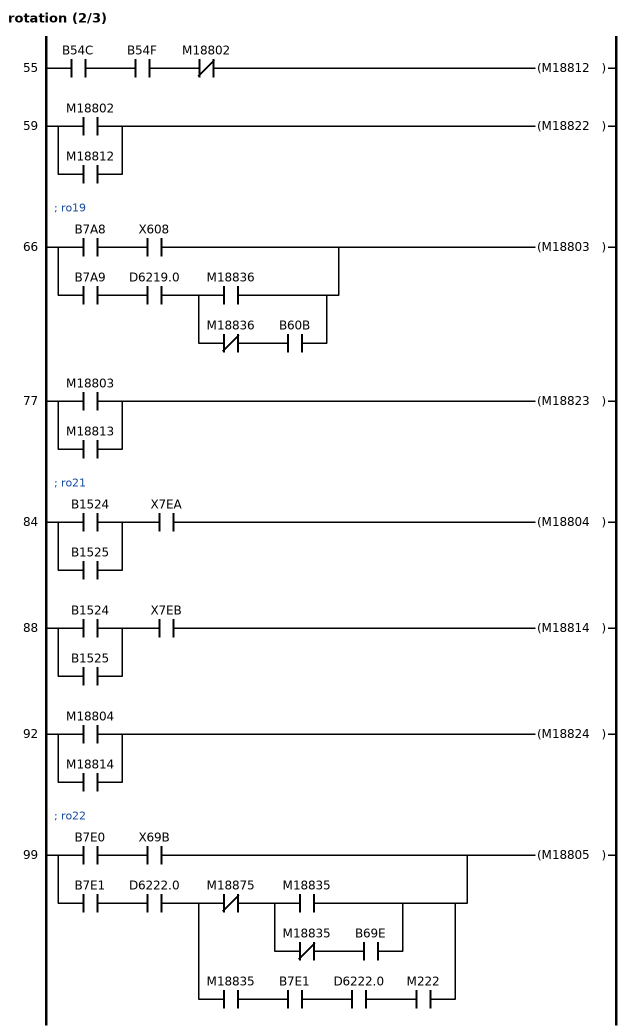
55    LD      B54C
      AND     B54F
      ANI     M18802
      OUT     M18812
59    LD      M18802
      OR      M18812
      OUT     M18822
; ro19
66    LD      B7A8
      AND     X608
      LD      B7A9
      AND     D6219.0
      LD      M18836
      LDI     M18836
      AND     B60B
      ORB
      ANB
      ORB
      OUT     M18803
77    LD      M18803
      OR      M18813
      OUT     M18823
; ro21
84    LD      B1524
      OR      B1525
      AND     X7EA
      OUT     M18804
88    LD      B1524
      OR      B1525
      AND     X7EB
      OUT     M18814
92    LD      M18804
      OR      M18814
      OUT     M18824
; ro22
99    LD      B7E0
      AND     X69B
      LD      B7E1
      AND     D6222.0
      LDI     M18875
      LD      M18835
      LDI     M18835
      AND     B69E
      ORB
      ANB
      LD      M18835
      AND     B7E1
      AND     D6222.0
      AND     M222
      ORB
      ANB
      ORB
      OUT     M18805
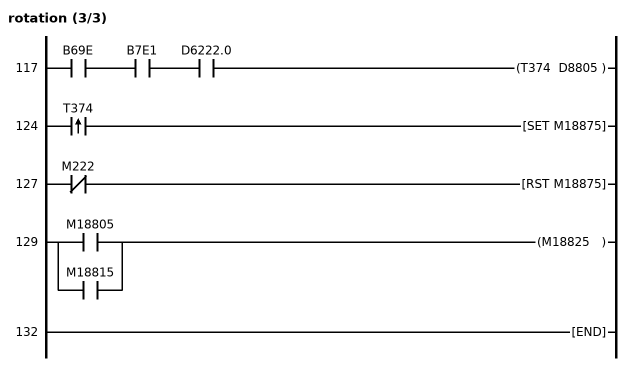
117   LD      B69E
      AND     B7E1
      AND     D6222.0
      OUT     T374 D8805
124   LDP     T374
      SET     M18875
127   LDI     M222
      RST     M18875
129   LD      M18805
      OR      M18815
      OUT     M18825
132   END
END_PROGRAM

PROGRAM safty
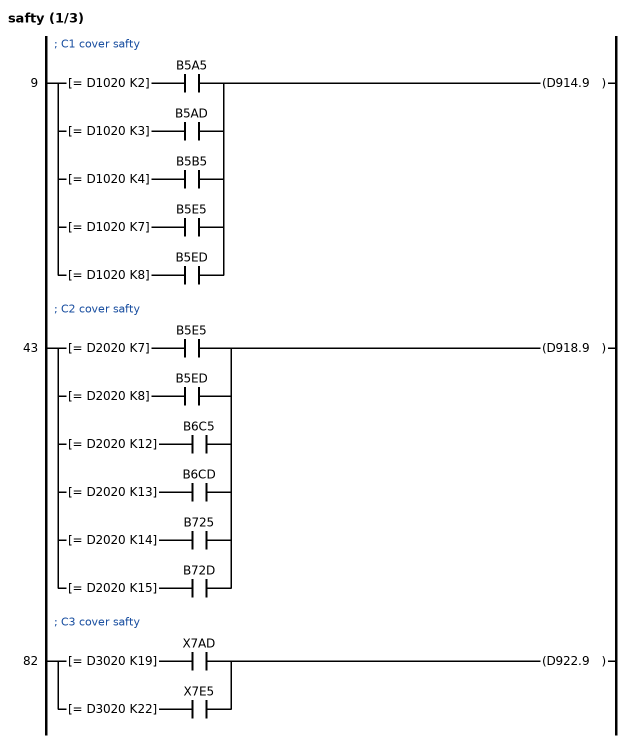
; C1 cover safty
9     LD=     D1020 K2
      AND     B5A5
      LD=     D1020 K3
      AND     B5AD
      ORB
      LD=     D1020 K4
      AND     B5B5
      ORB
      LD=     D1020 K7
      AND     B5E5
      ORB
      LD=     D1020 K8
      AND     B5ED
      ORB
      OUT     D914.9
; C2 cover safty
43    LD=     D2020 K7
      AND     B5E5
      LD=     D2020 K8
      AND     B5ED
      ORB
      LD=     D2020 K12
      AND     B6C5
      ORB
      LD=     D2020 K13
      AND     B6CD
      ORB
      LD=     D2020 K14
      AND     B725
      ORB
      LD=     D2020 K15
      AND     B72D
      ORB
      OUT     D918.9
; C3 cover safty
82    LD=     D3020 K19
      AND     X7AD
      LD=     D3020 K22
      AND     X7E5
      ORB
      OUT     D922.9
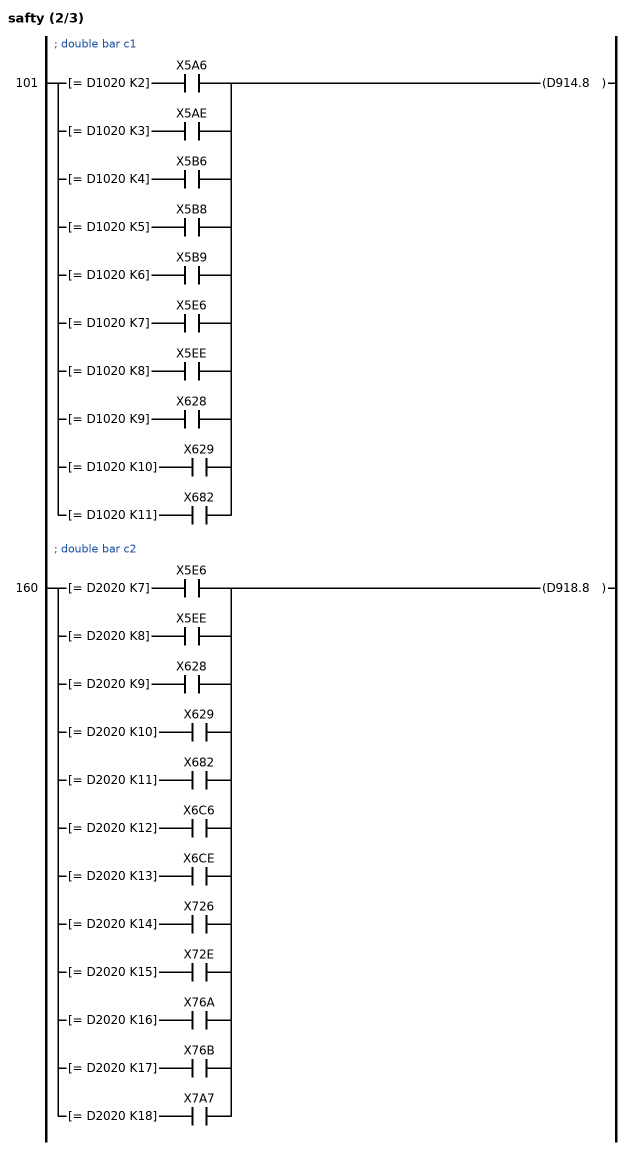
; double bar c1
101   LD=     D1020 K2
      AND     X5A6
      LD=     D1020 K3
      AND     X5AE
      ORB
      LD=     D1020 K4
      AND     X5B6
      ORB
      LD=     D1020 K5
      AND     X5B8
      ORB
      LD=     D1020 K6
      AND     X5B9
      ORB
      LD=     D1020 K7
      AND     X5E6
      ORB
      LD=     D1020 K8
      AND     X5EE
      ORB
      LD=     D1020 K9
      AND     X628
      ORB
      LD=     D1020 K10
      AND     X629
      ORB
      LD=     D1020 K11
      AND     X682
      ORB
      OUT     D914.8
; double bar c2
160   LD=     D2020 K7
      AND     X5E6
      LD=     D2020 K8
      AND     X5EE
      ORB
      LD=     D2020 K9
      AND     X628
      ORB
      LD=     D2020 K10
      AND     X629
      ORB
      LD=     D2020 K11
      AND     X682
      ORB
      LD=     D2020 K12
      AND     X6C6
      ORB
      LD=     D2020 K13
      AND     X6CE
      ORB
      LD=     D2020 K14
      AND     X726
      ORB
      LD=     D2020 K15
      AND     X72E
      ORB
      LD=     D2020 K16
      AND     X76A
      ORB
      LD=     D2020 K17
      AND     X76B
      ORB
      LD=     D2020 K18
      AND     X7A7
      ORB
      OUT     D918.8
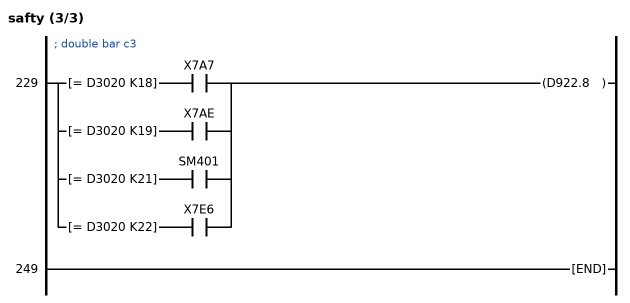
; double bar c3
229   LD=     D3020 K18
      AND     X7A7
      LD=     D3020 K19
      AND     X7AE
      ORB
      LD=     D3020 K21
      AND     SM401
      ORB
      LD=     D3020 K22
      AND     X7E6
      ORB
      OUT     D922.8
249   END
END_PROGRAM

PROGRAM Scrubber
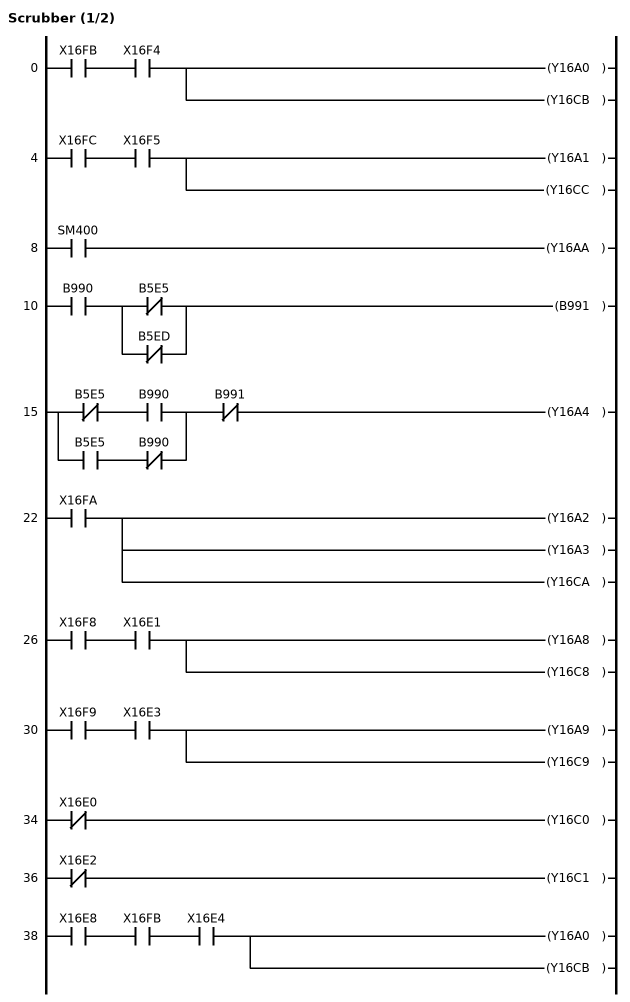
0     LD      X16FB
      AND     X16F4
      OUT     Y16A0
      OUT     Y16CB
4     LD      X16FC
      AND     X16F5
      OUT     Y16A1
      OUT     Y16CC
8     LD      SM400
      OUT     Y16AA
10    LD      B990
      LDI     B5E5
      ORI     B5ED
      ANB
      OUT     B991
15    LDI     B5E5
      AND     B990
      LD      B5E5
      ANI     B990
      ORB
      ANI     B991
      OUT     Y16A4
22    LD      X16FA
      OUT     Y16A2
      OUT     Y16A3
      OUT     Y16CA
26    LD      X16F8
      AND     X16E1
      OUT     Y16A8
      OUT     Y16C8
30    LD      X16F9
      AND     X16E3
      OUT     Y16A9
      OUT     Y16C9
34    LDI     X16E0
      OUT     Y16C0
36    LDI     X16E2
      OUT     Y16C1
38    LD      X16E8
      AND     X16FB
      AND     X16E4
      OUT     Y16A0
      OUT     Y16CB
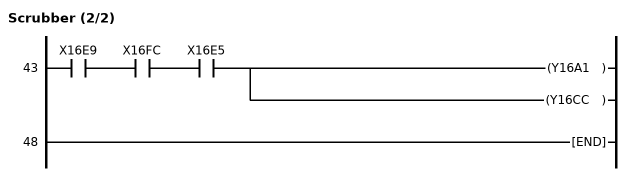
43    LD      X16E9
      AND     X16FC
      AND     X16E5
      OUT     Y16A1
      OUT     Y16CC
48    END
END_PROGRAM

PROGRAM send_to_c
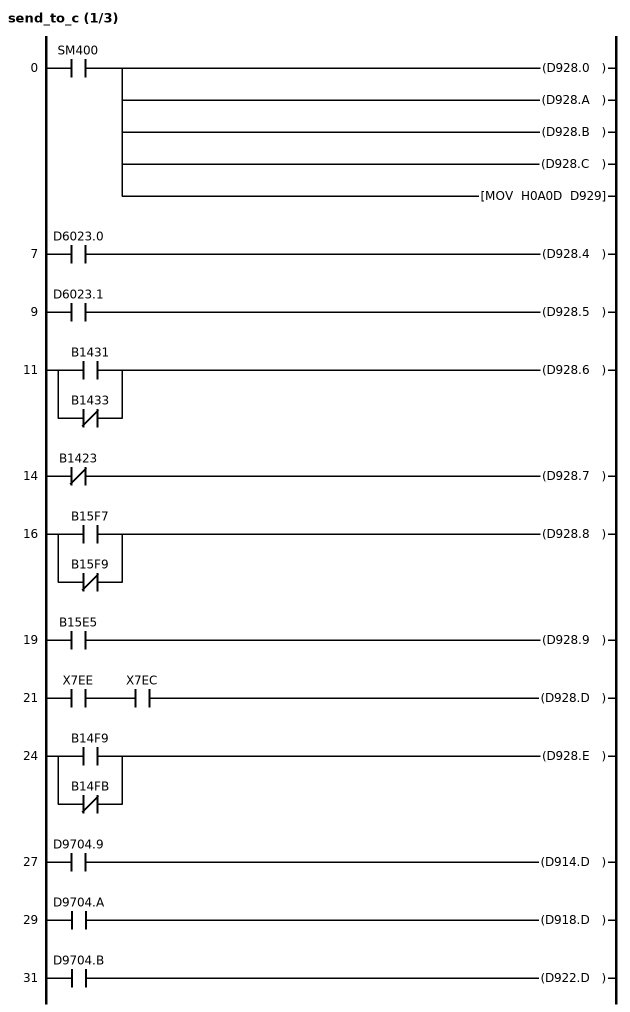
0     LD      SM400
      OUT     D928.0
      OUT     D928.A
      OUT     D928.B
      OUT     D928.C
      MOV     H0A0D D929
7     LD      D6023.0
      OUT     D928.4
9     LD      D6023.1
      OUT     D928.5
11    LD      B1431
      ORI     B1433
      OUT     D928.6
14    LDI     B1423
      OUT     D928.7
16    LD      B15F7
      ORI     B15F9
      OUT     D928.8
19    LD      B15E5
      OUT     D928.9
21    LD      X7EE
      AND     X7EC
      OUT     D928.D
24    LD      B14F9
      ORI     B14FB
      OUT     D928.E
27    LD      D9704.9
      OUT     D914.D
29    LD      D9704.A
      OUT     D918.D
31    LD      D9704.B
      OUT     D922.D
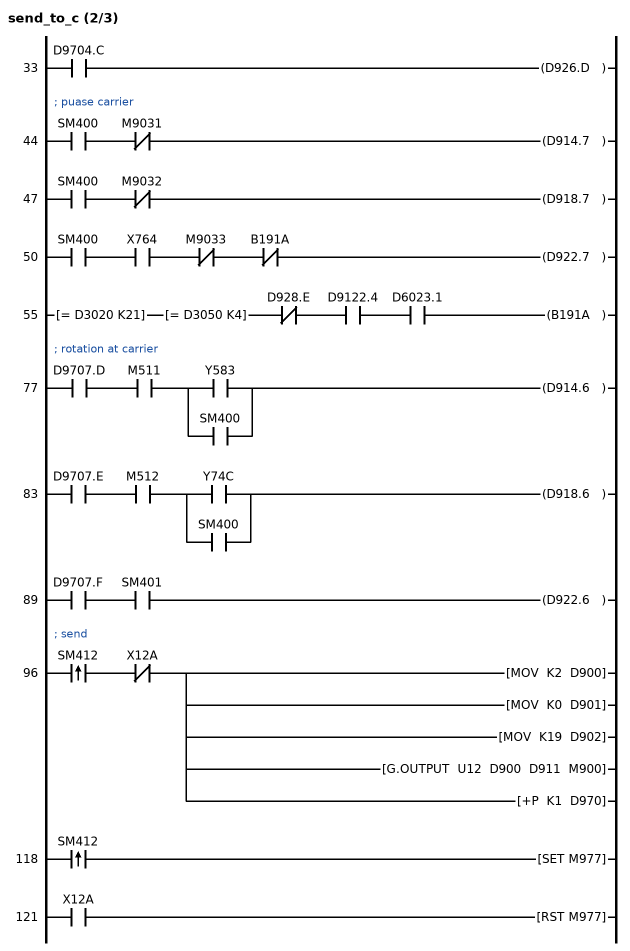
33    LD      D9704.C
      OUT     D926.D
; puase carrier
44    LD      SM400
      ANI     M9031
      OUT     D914.7
47    LD      SM400
      ANI     M9032
      OUT     D918.7
50    LD      SM400
      AND     X764
      ANI     M9033
      ANI     B191A
      OUT     D922.7
55    LD=     D3020 K21
      AND=    D3050 K4
      ANI     D928.E
      AND     D9122.4
      AND     D6023.1
      OUT     B191A
; rotation at carrier
77    LD      D9707.D
      AND     M511
      LD      Y583
      OR      SM400
      ANB
      OUT     D914.6
83    LD      D9707.E
      AND     M512
      LD      Y74C
      OR      SM400
      ANB
      OUT     D918.6
89    LD      D9707.F
      AND     SM401
      OUT     D922.6
; send
96    LDP     SM412
      ANI     X12A
      MOV     K2 D900
      MOV     K0 D901
      MOV     K19 D902
      G.OUTPUT U12 D900 D911 M900
      +P      K1 D970
118   LDP     SM412
      SET     M977
121   LD      X12A
      RST     M977
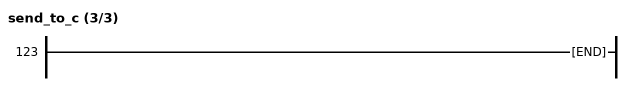
123   END
END_PROGRAM

PROGRAM sent_to_c_key
VAR
  __IST_9118b3cfc5d74fe4 : I+ST_9118b3cfc5d74fe4;
END_VAR
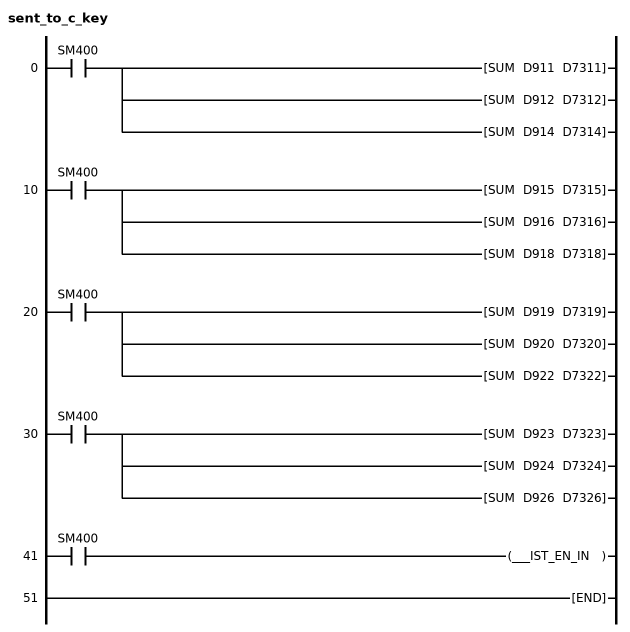
0     LD      SM400
      SUM     D911 D7311
      SUM     D912 D7312
      SUM     D914 D7314
10    LD      SM400
      SUM     D915 D7315
      SUM     D916 D7316
      SUM     D918 D7318
20    LD      SM400
      SUM     D919 D7319
      SUM     D920 D7320
      SUM     D922 D7322
30    LD      SM400
      SUM     D923 D7323
      SUM     D924 D7324
      SUM     D926 D7326
; FB BLK START I+ST_9118b3cfc5d74fe4(__IST_9118b3cfc5d74fe4)
41    LD      SM400
      OUT     ___IST_EN_IN
; FB START
; FB_NAME I+ST_9118b3cfc5d74fe4
; INSTANCE_NAME __IST_9118b3cfc5d74fe4
; FB IN_B:__IST_EN_IN
; FB OUT___IST_EN_OUT:B
; FB END
; FB BLK END
51    END
END_PROGRAM

PROGRAM shower
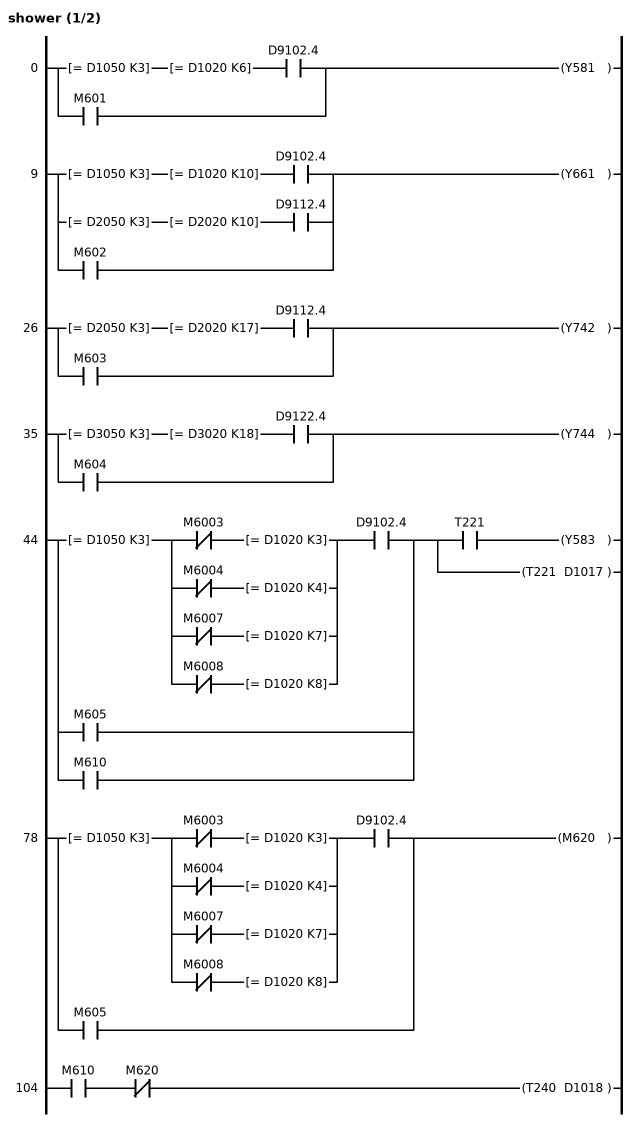
0     LD=     D1050 K3
      AND=    D1020 K6
      AND     D9102.4
      OR      M601
      OUT     Y581
9     LD=     D1050 K3
      AND=    D1020 K10
      AND     D9102.4
      LD=     D2050 K3
      AND=    D2020 K10
      AND     D9112.4
      ORB
      OR      M602
      OUT     Y661
26    LD=     D2050 K3
      AND=    D2020 K17
      AND     D9112.4
      OR      M603
      OUT     Y742
35    LD=     D3050 K3
      AND=    D3020 K18
      AND     D9122.4
      OR      M604
      OUT     Y744
44    LD=     D1050 K3
      LDI     M6003
      AND=    D1020 K3
      LDI     M6004
      AND=    D1020 K4
      ORB
      LDI     M6007
      AND=    D1020 K7
      ORB
      LDI     M6008
      AND=    D1020 K8
      ORB
      ANB
      AND     D9102.4
      OR      M605
      OR      M610
      MPS
      AND     T221
      OUT     Y583
      MPP
      OUT     T221 D1017
78    LD=     D1050 K3
      LDI     M6003
      AND=    D1020 K3
      LDI     M6004
      AND=    D1020 K4
      ORB
      LDI     M6007
      AND=    D1020 K7
      ORB
      LDI     M6008
      AND=    D1020 K8
      ORB
      ANB
      AND     D9102.4
      OR      M605
      OUT     M620
104   LD      M610
      ANI     M620
      OUT     T240 D1018
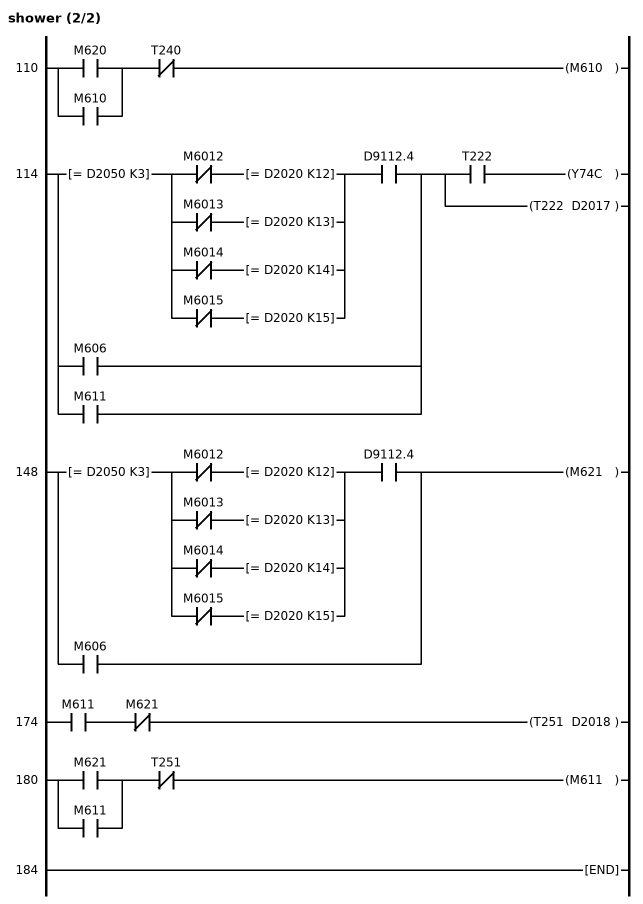
110   LD      M620
      OR      M610
      ANI     T240
      OUT     M610
114   LD=     D2050 K3
      LDI     M6012
      AND=    D2020 K12
      LDI     M6013
      AND=    D2020 K13
      ORB
      LDI     M6014
      AND=    D2020 K14
      ORB
      LDI     M6015
      AND=    D2020 K15
      ORB
      ANB
      AND     D9112.4
      OR      M606
      OR      M611
      MPS
      AND     T222
      OUT     Y74C
      MPP
      OUT     T222 D2017
148   LD=     D2050 K3
      LDI     M6012
      AND=    D2020 K12
      LDI     M6013
      AND=    D2020 K13
      ORB
      LDI     M6014
      AND=    D2020 K14
      ORB
      LDI     M6015
      AND=    D2020 K15
      ORB
      ANB
      AND     D9112.4
      OR      M606
      OUT     M621
174   LD      M611
      ANI     M621
      OUT     T251 D2018
180   LD      M621
      OR      M611
      ANI     T251
      OUT     M611
184   END
END_PROGRAM

FUNCTION_BLOCK tank_PV
VAR_INPUT
  ON_BY_ORDER : BOOL;
  Stay_ON : BOOL;
  Reset_0 : BOOL;
END_VAR
VAR_OUTPUT
  PV : INT;
END_VAR
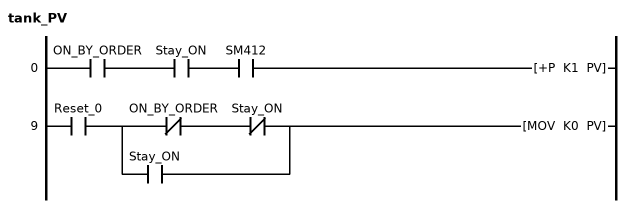
0     LD      ON_BY_ORDER
      AND     Stay_ON
      AND     SM412
      +P      K1 PV
9     LD      Reset_0
      LDI     ON_BY_ORDER
      ANI     Stay_ON
      OR      Stay_ON
      ANB
      MOV     K0 PV
END_FUNCTION_BLOCK

PROGRAM tank_time_B
VAR
  tank_PV_202 : tank_PV;
  tank_PV_203 : tank_PV;
  tank_PV_204 : tank_PV;
  tank_PV_205 : tank_PV;
  tank_PV_206 : tank_PV;
  tank_PV_207 : tank_PV;
  tank_PV_208 : tank_PV;
  tank_PV_209 : tank_PV;
  tank_PV_210 : tank_PV;
  tank_PV_211 : tank_PV;
  tank_PV_212 : tank_PV;
  tank_PV_213 : tank_PV;
  tank_PV_214 : tank_PV;
  tank_PV_215 : tank_PV;
  tank_PV_216 : tank_PV;
  tank_PV_217 : tank_PV;
  tank_PV_218 : tank_PV;
  tank_PV_219 : tank_PV;
  tank_PV_221 : tank_PV;
  tank_PV_222 : tank_PV;
END_VAR
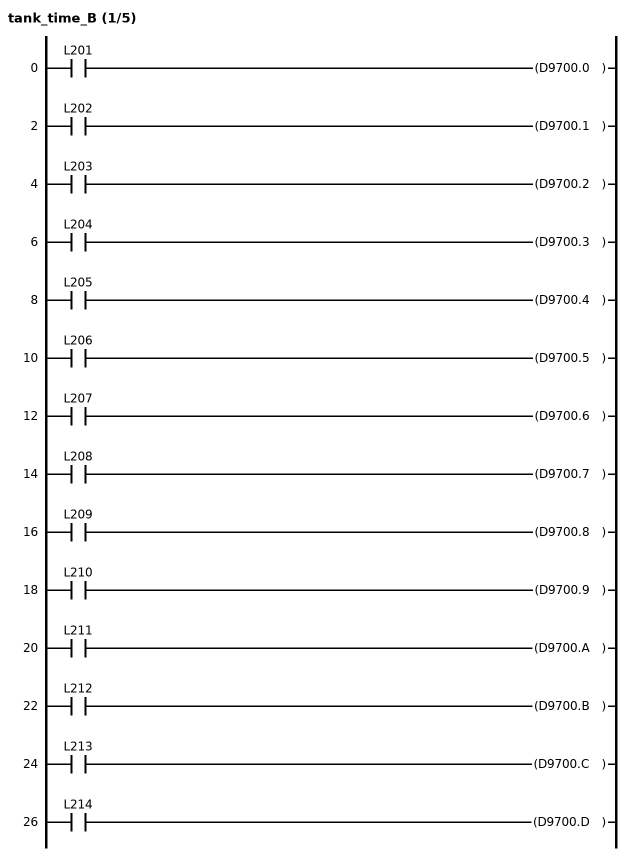
0     LD      L201
      OUT     D9700.0
2     LD      L202
      OUT     D9700.1
4     LD      L203
      OUT     D9700.2
6     LD      L204
      OUT     D9700.3
8     LD      L205
      OUT     D9700.4
10    LD      L206
      OUT     D9700.5
12    LD      L207
      OUT     D9700.6
14    LD      L208
      OUT     D9700.7
16    LD      L209
      OUT     D9700.8
18    LD      L210
      OUT     D9700.9
20    LD      L211
      OUT     D9700.A
22    LD      L212
      OUT     D9700.B
24    LD      L213
      OUT     D9700.C
26    LD      L214
      OUT     D9700.D
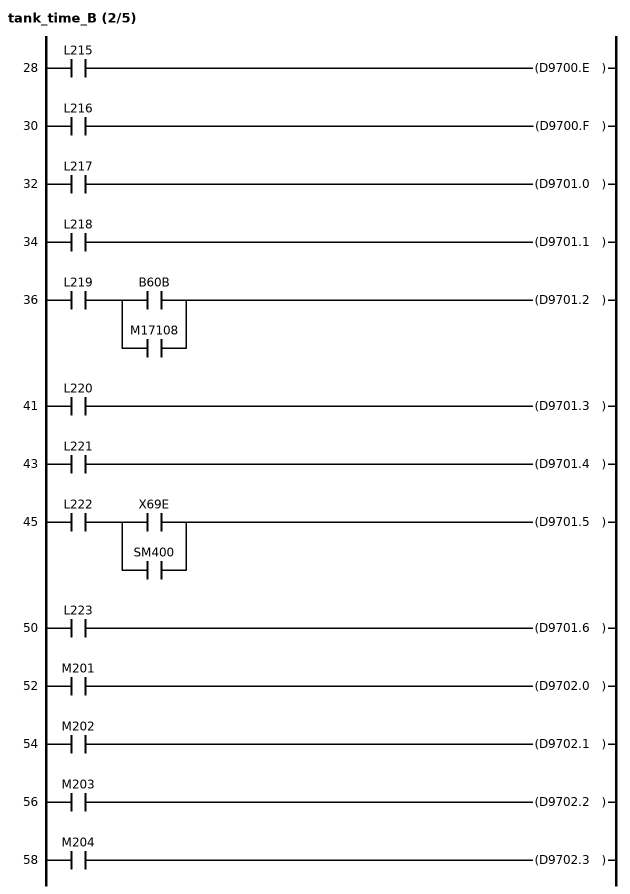
28    LD      L215
      OUT     D9700.E
30    LD      L216
      OUT     D9700.F
32    LD      L217
      OUT     D9701.0
34    LD      L218
      OUT     D9701.1
36    LD      L219
      LD      B60B
      OR      M17108
      ANB
      OUT     D9701.2
41    LD      L220
      OUT     D9701.3
43    LD      L221
      OUT     D9701.4
45    LD      L222
      LD      X69E
      OR      SM400
      ANB
      OUT     D9701.5
50    LD      L223
      OUT     D9701.6
52    LD      M201
      OUT     D9702.0
54    LD      M202
      OUT     D9702.1
56    LD      M203
      OUT     D9702.2
58    LD      M204
      OUT     D9702.3
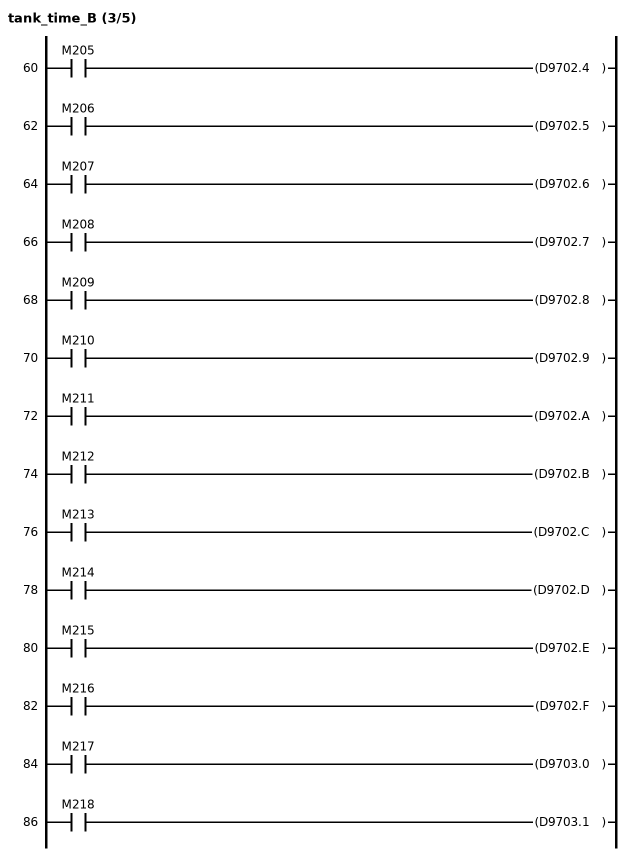
60    LD      M205
      OUT     D9702.4
62    LD      M206
      OUT     D9702.5
64    LD      M207
      OUT     D9702.6
66    LD      M208
      OUT     D9702.7
68    LD      M209
      OUT     D9702.8
70    LD      M210
      OUT     D9702.9
72    LD      M211
      OUT     D9702.A
74    LD      M212
      OUT     D9702.B
76    LD      M213
      OUT     D9702.C
78    LD      M214
      OUT     D9702.D
80    LD      M215
      OUT     D9702.E
82    LD      M216
      OUT     D9702.F
84    LD      M217
      OUT     D9703.0
86    LD      M218
      OUT     D9703.1
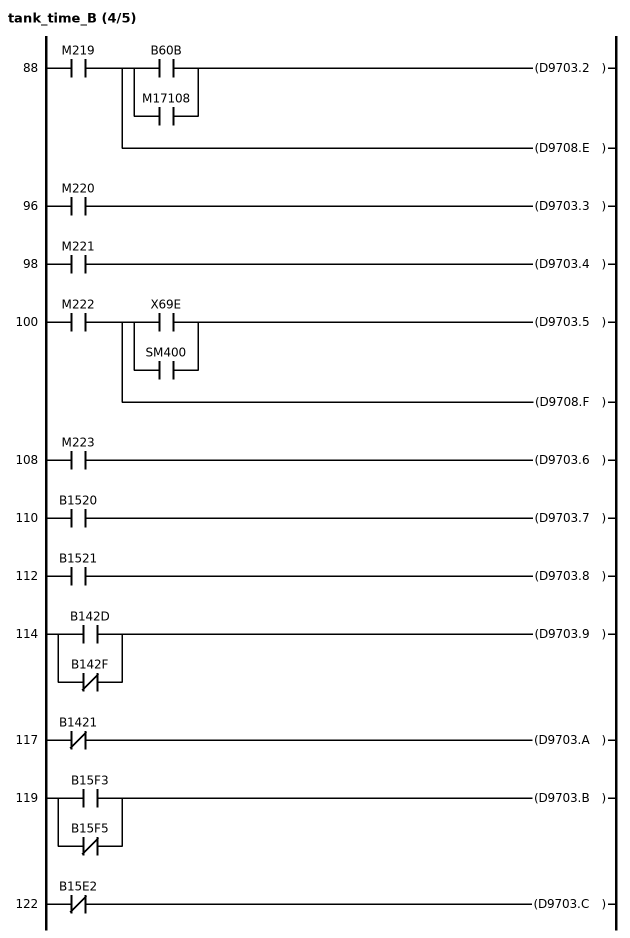
88    LD      M219
      MPS
      LD      B60B
      OR      M17108
      ANB
      OUT     D9703.2
      MPP
      OUT     D9708.E
96    LD      M220
      OUT     D9703.3
98    LD      M221
      OUT     D9703.4
100   LD      M222
      MPS
      LD      X69E
      OR      SM400
      ANB
      OUT     D9703.5
      MPP
      OUT     D9708.F
108   LD      M223
      OUT     D9703.6
110   LD      B1520
      OUT     D9703.7
112   LD      B1521
      OUT     D9703.8
114   LD      B142D
      ORI     B142F
      OUT     D9703.9
117   LDI     B1421
      OUT     D9703.A
119   LD      B15F3
      ORI     B15F5
      OUT     D9703.B
122   LDI     B15E2
      OUT     D9703.C
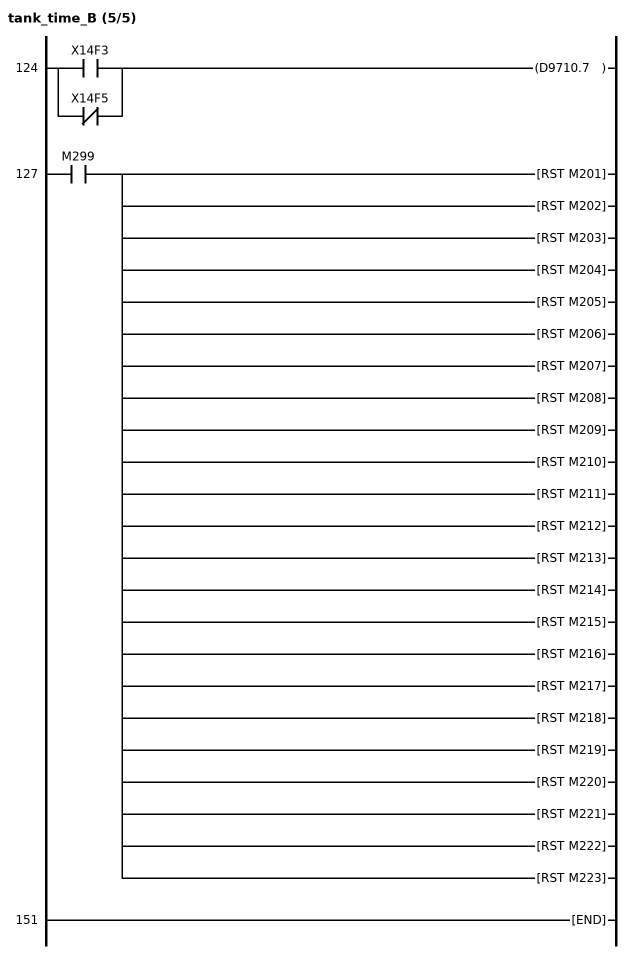
124   LD      X14F3
      ORI     X14F5
      OUT     D9710.7
127   LD      M299
      RST     M201
      RST     M202
      RST     M203
      RST     M204
      RST     M205
      RST     M206
      RST     M207
      RST     M208
      RST     M209
      RST     M210
      RST     M211
      RST     M212
      RST     M213
      RST     M214
      RST     M215
      RST     M216
      RST     M217
      RST     M218
      RST     M219
      RST     M220
      RST     M221
      RST     M222
      RST     M223
151   END
END_PROGRAM

PROGRAM temp_system
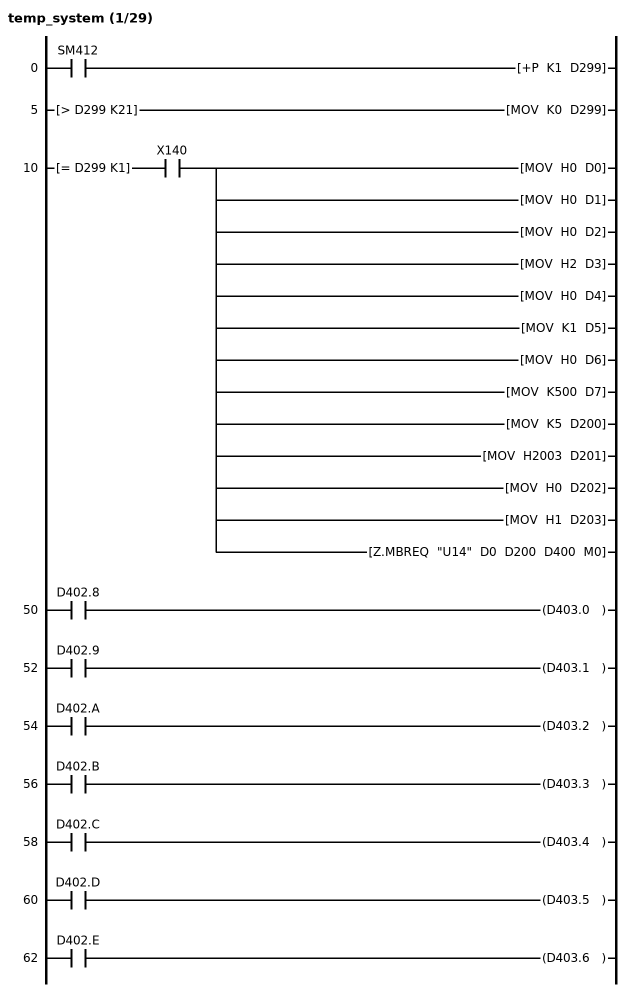
0     LD      SM412
      +P      K1 D299
5     LD>     D299 K21
      MOV     K0 D299
10    LD=     D299 K1
      AND     X140
      MOV     H0 D0
      MOV     H0 D1
      MOV     H0 D2
      MOV     H2 D3
      MOV     H0 D4
      MOV     K1 D5
      MOV     H0 D6
      MOV     K500 D7
      MOV     K5 D200
      MOV     H2003 D201
      MOV     H0 D202
      MOV     H1 D203
      Z.MBREQ "U14" D0 D200 D400 M0
50    LD      D402.8
      OUT     D403.0
52    LD      D402.9
      OUT     D403.1
54    LD      D402.A
      OUT     D403.2
56    LD      D402.B
      OUT     D403.3
58    LD      D402.C
      OUT     D403.4
60    LD      D402.D
      OUT     D403.5
62    LD      D402.E
      OUT     D403.6
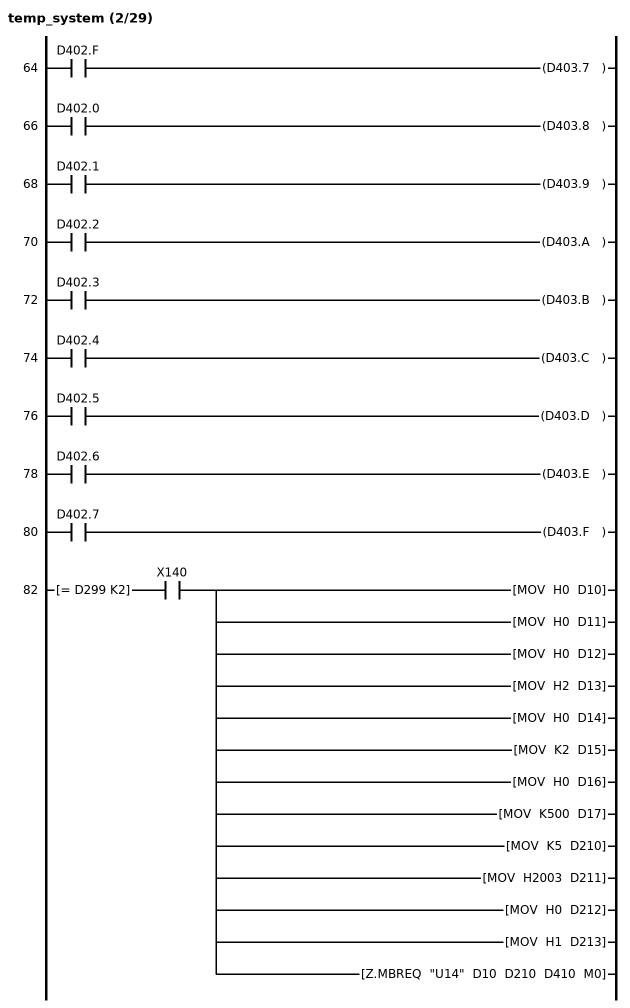
64    LD      D402.F
      OUT     D403.7
66    LD      D402.0
      OUT     D403.8
68    LD      D402.1
      OUT     D403.9
70    LD      D402.2
      OUT     D403.A
72    LD      D402.3
      OUT     D403.B
74    LD      D402.4
      OUT     D403.C
76    LD      D402.5
      OUT     D403.D
78    LD      D402.6
      OUT     D403.E
80    LD      D402.7
      OUT     D403.F
82    LD=     D299 K2
      AND     X140
      MOV     H0 D10
      MOV     H0 D11
      MOV     H0 D12
      MOV     H2 D13
      MOV     H0 D14
      MOV     K2 D15
      MOV     H0 D16
      MOV     K500 D17
      MOV     K5 D210
      MOV     H2003 D211
      MOV     H0 D212
      MOV     H1 D213
      Z.MBREQ "U14" D10 D210 D410 M0
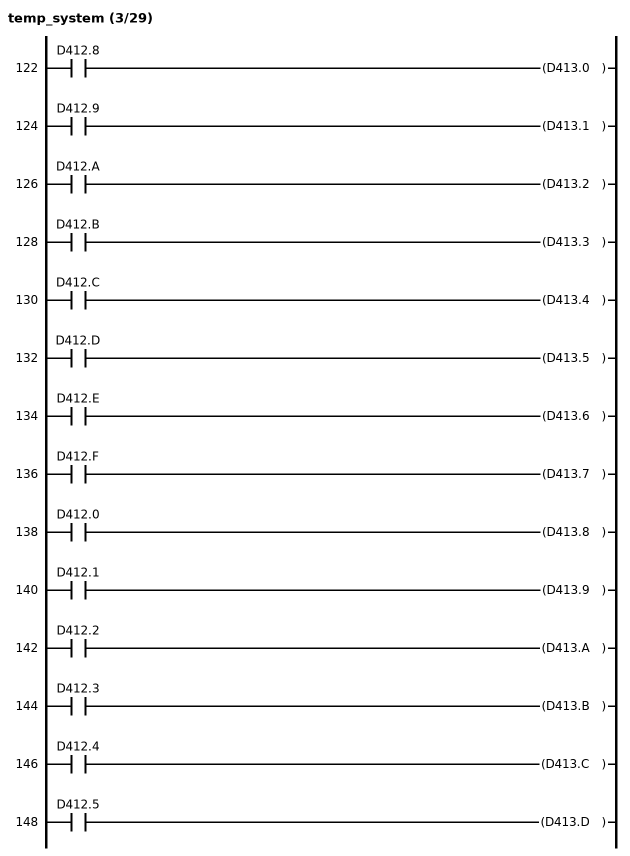
122   LD      D412.8
      OUT     D413.0
124   LD      D412.9
      OUT     D413.1
126   LD      D412.A
      OUT     D413.2
128   LD      D412.B
      OUT     D413.3
130   LD      D412.C
      OUT     D413.4
132   LD      D412.D
      OUT     D413.5
134   LD      D412.E
      OUT     D413.6
136   LD      D412.F
      OUT     D413.7
138   LD      D412.0
      OUT     D413.8
140   LD      D412.1
      OUT     D413.9
142   LD      D412.2
      OUT     D413.A
144   LD      D412.3
      OUT     D413.B
146   LD      D412.4
      OUT     D413.C
148   LD      D412.5
      OUT     D413.D
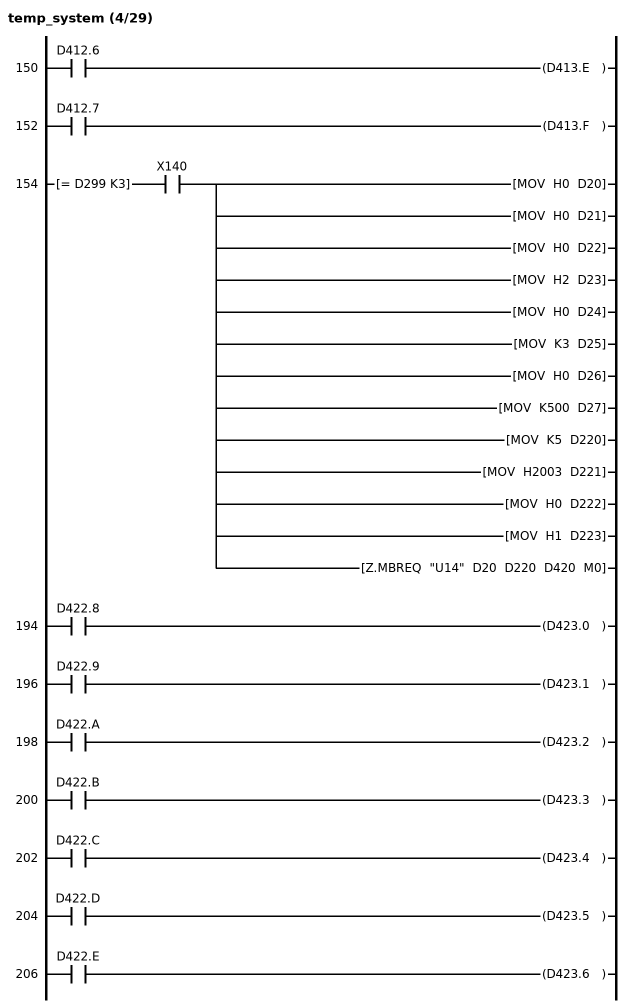
150   LD      D412.6
      OUT     D413.E
152   LD      D412.7
      OUT     D413.F
154   LD=     D299 K3
      AND     X140
      MOV     H0 D20
      MOV     H0 D21
      MOV     H0 D22
      MOV     H2 D23
      MOV     H0 D24
      MOV     K3 D25
      MOV     H0 D26
      MOV     K500 D27
      MOV     K5 D220
      MOV     H2003 D221
      MOV     H0 D222
      MOV     H1 D223
      Z.MBREQ "U14" D20 D220 D420 M0
194   LD      D422.8
      OUT     D423.0
196   LD      D422.9
      OUT     D423.1
198   LD      D422.A
      OUT     D423.2
200   LD      D422.B
      OUT     D423.3
202   LD      D422.C
      OUT     D423.4
204   LD      D422.D
      OUT     D423.5
206   LD      D422.E
      OUT     D423.6
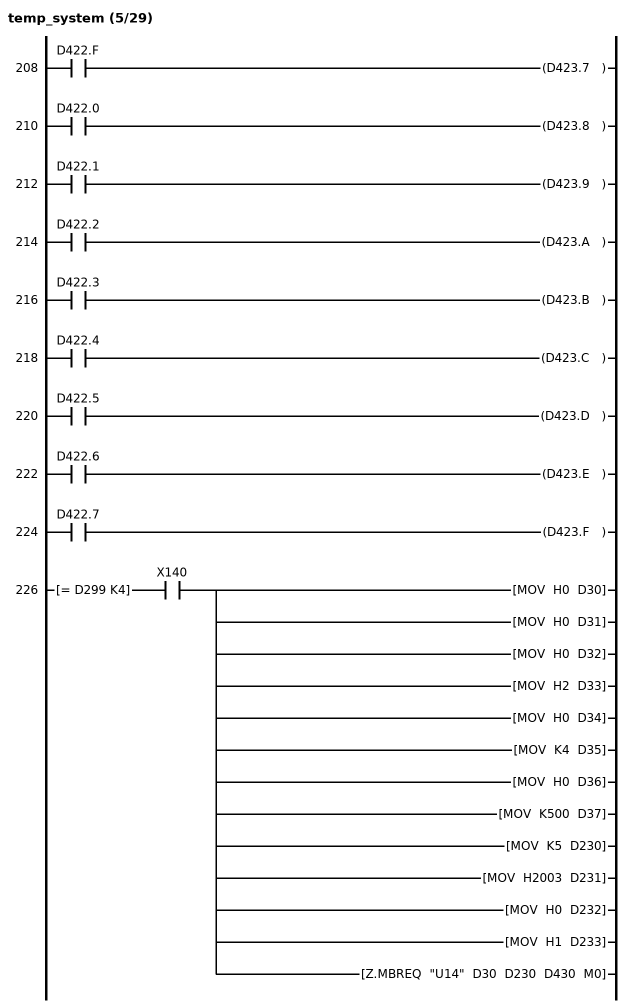
208   LD      D422.F
      OUT     D423.7
210   LD      D422.0
      OUT     D423.8
212   LD      D422.1
      OUT     D423.9
214   LD      D422.2
      OUT     D423.A
216   LD      D422.3
      OUT     D423.B
218   LD      D422.4
      OUT     D423.C
220   LD      D422.5
      OUT     D423.D
222   LD      D422.6
      OUT     D423.E
224   LD      D422.7
      OUT     D423.F
226   LD=     D299 K4
      AND     X140
      MOV     H0 D30
      MOV     H0 D31
      MOV     H0 D32
      MOV     H2 D33
      MOV     H0 D34
      MOV     K4 D35
      MOV     H0 D36
      MOV     K500 D37
      MOV     K5 D230
      MOV     H2003 D231
      MOV     H0 D232
      MOV     H1 D233
      Z.MBREQ "U14" D30 D230 D430 M0
